Universal Robots PolyScope program: mt.urp

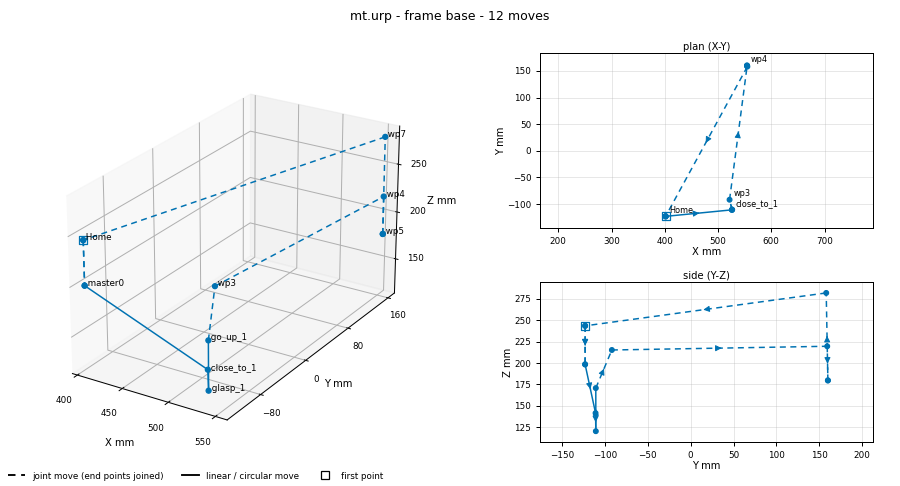
[picture p0: tool path of mt.urp in frame base, 12 of 12 moves have a stored position in this frame; points joined in program order, loops and branches not executed]
Program mt (installation=default directory=/programs/rovi createdIn=3.8.0.61336 lastSavedIn=3.8.0.61336 robotSerialNumber=2016352774)
Calibrated DH parameters: a=[0.000165, -0.326475, -0.363587, -0.000196, 0.000314, 0]; d=[0.089242, 611.192012, -553.715229, -57.366527, 0.094858, 0.082351]; alpha=[1.570545, 0.000446, 0.002569, 1.569839, -1.569769, 0]; deltaTheta=[-0.000028, 0.695517, -0.309849, -0.385645, -0.000052, -0.000026]
Robot Program (runOnlyOnce=false)
  MoveJ speed 60 deg/s, acceleration 80 deg/s^2 (useActiveTCP=false)
    Waypoint Home: TCP in base x=401.617 y=-123.055 z=243.432 mm, rx=-0.302 ry=3.1208 rz=0.0289 rad; joints [-1.945, -85.366, -123.205, -61.282, 91.24, -13.048] deg; flange x=401.666 y=-123.045 z=243.433 mm, rx=-2.4115 ry=1.9862 rz=0.0137 rad
  Loop Forever
    Script file /programs/X0.script
      | address="172.16.58.34"
      | port=3000
      | socket_open(address,port)
      | socket_send_line("X0()")
      | ret=socket_read_line(timeout=3)
      | socket_close()
    SuppressedNode
      MoveJ speed 60 deg/s, acceleration 80 deg/s^2 (useActiveTCP=false)
        Waypoint capture0: TCP in base x=291.074 y=-404.604 z=201.943 mm, rx=-1.3664 ry=-2.7229 rz=0.0094 rad; joints [-41.118, -99.563, -113.852, -61.83, 88.448, 12.2] deg
    MoveJ speed 60 deg/s, acceleration 80 deg/s^2 (useActiveTCP=false)
      Waypoint master0: TCP in base x=401.618 y=-123.109 z=198.453 mm, rx=-0.3017 ry=3.1209 rz=0.0292 rad; joints [-1.958, -89.361, -127.245, -53.252, 91.245, -13.033] deg; flange x=401.667 y=-123.1 z=198.454 mm, rx=-2.4113 ry=1.9864 rz=0.0139 rad
      Wait Sleep waitTime=0.5
    X_error := True
    Loop While (checkContinuously=false) expression=X_error
      Loop While (checkContinuously=false) expression=X_error
        Script file /programs/X1.script
          | address="172.16.58.34"
          | port=3000
          | X_error=False
          | socket_open(address,port)
          | p=get_actual_tcp_pose()
          | rpy=rotvec2rpy([p[3],p[4],p[5]])
          | socket_send_string("X1(")
          | socket_send_string(p[0])
          | socket_send_string(",")
          | socket_send_string(p[1])
          | socket_send_string(",")
          | socket_send_string(p[2])
          | socket_send_string(",")
          | socket_send_string(r2d(rpy[0]))
          | socket_send_string(",")
          | socket_send_string(r2d(rpy[1]))
          | socket_send_string(",")
          | socket_send_string(r2d(rpy[2]))
          | socket_send_line(")")
          | ret=socket_read_line(timeout=10)
          | if (ret!="OK"):
          |   X_error=True
          |   code=socket_read_string()
          |   popup(code,title="X1",blocking=True)
          | end
          | socket_close()
        Wait Sleep waitTime=0.5
      Script file /programs/rovi/X2.script
        | global X_var=Base
        | address="172.16.58.34"
        | port=3000
        | X_error=False
        | socket_open(address,port)
        | socket_send_line("X2()")
        | ret=socket_read_line(timeout=10)
        | if (ret != "OK"):
        |   X_error=True
        |   socket_close()
        | else:
        |   f=socket_read_ascii_float(6)
        |   while (f[0]!=6):
        |     sleep(0.3)
        |     f=socket_read_ascii_float(6)
        |   end
        |   socket_close()
        |   #popup(f,title="OK",blocking=True)
        |   rvec=rpy2rotvec([d2r(f[4]),d2r(f[5]),d2r(f[6])])
        |   counter=0
        |   while (counter<3):
        |     X_var[counter]=f[counter+1]
        |     counter=counter+1
        |   end
        |   counter=0
        |   while (counter<3):
        |     X_var[counter+3]=rvec[counter]
        |     counter=counter+1
        |   end
        | end
    Base := X_var
    MoveL speed 250 mm/s, acceleration 1200 mm/s^2 (useActiveTCP=false) feature(featureName=Joint_0_name)
      Waypoint close_to_1: TCP in base x=525.892 y=-110.922 z=141.644 mm, rx=-0.0249 ry=3.1389 rz=0.0305 rad; joints [-0.174, -109.589, -113.105, -47.241, 91.26, -1.103] deg; flange x=525.942 y=-110.921 z=141.644 mm, rx=-2.2278 ry=2.193 rz=0.0188 rad
      Waypoint glasp_1: TCP in base x=526.359 y=-110.603 z=120.526 mm, rx=-0.0225 ry=3.1387 rz=0.0305 rad; joints [-0.14, -111.796, -114.027, -44.096, 91.259, -0.976] deg
      Waypoint go_up_1: TCP in base x=526.461 y=-110.629 z=170.827 mm, rx=-0.0309 ry=3.1386 rz=0.0301 rad; joints [-0.138, -106.888, -111.412, -51.62, 91.249, -1.298] deg; flange x=526.511 y=-110.628 z=170.827 mm, rx=-2.232 ry=2.1887 rz=0.0182 rad
    MoveJ speed 60 deg/s, acceleration 80 deg/s^2 (useActiveTCP=false)
      Waypoint wp3: TCP in base x=521.639 y=-91.889 z=215.25 mm, rx=0.1315 ry=-3.1327 rz=-0.029 rad; joints [1.934, -102.24, -109.536, -58.64, 91.208, -2.926] deg; flange x=521.689 y=-91.885 z=215.25 mm, rx=-2.306 ry=2.1204 rz=0.0272 rad
      Waypoint wp4: TCP in base x=554.629 y=159.317 z=219.592 mm, rx=0.0228 ry=-3.1347 rz=-0.0286 rad; joints [26.953, -107.73, -101.658, -60.547, 91.26, 26.066] deg; flange x=554.679 y=159.318 z=219.591 mm, rx=-2.2315 ry=2.1995 rz=0.0276 rad
      Waypoint wp5: TCP in base x=554.357 y=160.095 z=179.72 mm, rx=0.0229 ry=-3.1347 rz=-0.0286 rad; joints [27.033, -110.662, -104.375, -54.897, 91.26, 26.156] deg; flange x=554.407 y=160.096 z=179.72 mm, rx=-2.2316 ry=2.1994 rz=0.0276 rad
      Waypoint wp6: TCP in base x=554.363 y=160.071 z=179.768 mm, rx=0.0228 ry=-3.1348 rz=-0.0288 rad; joints [27.031, -110.657, -104.374, -54.896, 91.262, 26.159] deg; flange x=554.413 y=160.072 z=179.767 mm, rx=-2.2314 ry=2.1994 rz=0.0276 rad
      Waypoint wp7: TCP in base x=555.075 y=158.144 z=281.8 mm, rx=0.0225 ry=-3.1348 rz=-0.0287 rad; joints [26.83, -104.167, -96.365, -69.405, 91.26, 25.931] deg; flange x=555.125 y=158.145 z=281.8 mm, rx=-2.2313 ry=2.1997 rz=0.0276 rad
    MoveJ speed 60 deg/s, acceleration 80 deg/s^2 (useActiveTCP=false)
      Waypoint Home: TCP in base x=401.617 y=-123.055 z=243.432 mm, rx=-0.302 ry=3.1208 rz=0.0289 rad; joints [-1.945, -85.366, -123.205, -61.282, 91.24, -13.048] deg; flange x=401.666 y=-123.045 z=243.433 mm, rx=-2.4115 ry=1.9862 rz=0.0137 rad
  Halt
  Folder Manual operation
    MoveJ speed 60 deg/s, acceleration 80 deg/s^2 (useActiveTCP=false)
      Waypoint master0: TCP in base x=401.618 y=-123.109 z=198.453 mm, rx=-0.3017 ry=3.1209 rz=0.0292 rad; joints [-1.958, -89.361, -127.245, -53.252, 91.245, -13.033] deg; flange x=401.667 y=-123.1 z=198.454 mm, rx=-2.4113 ry=1.9864 rz=0.0139 rad
    Base := Base
    Script file /programs/rovi/X0.script
      | address="172.16.58.34"
      | port=3000
      | socket_open(address,port)
      | socket_send_line("X0()")
      | ret=socket_read_line(timeout=3)
      | socket_close()
      | Base=p[0,0,0,0,0,0]
    Script file /programs/rovi/X1.script
      | address="172.16.58.34"
      | port=3000
      | timeout=10
      | socket_open(address,port)
      | p=get_actual_tcp_pose()
      | rpy=rotvec2rpy([p[3],p[4],p[5]])
      | socket_send_string("X1(")
      | socket_send_string(p[0])
      | socket_send_string(",")
      | socket_send_string(p[1])
      | socket_send_string(",")
      | socket_send_string(p[2])
      | socket_send_string(",")
      | socket_send_string(r2d(rpy[0]))
      | socket_send_string(",")
      | socket_send_string(r2d(rpy[1]))
      | socket_send_string(",")
      | socket_send_string(r2d(rpy[2]))
      | socket_send_line(")")
      | ret=socket_read_line(timeout=10)
      | if (ret!="OK"):
      |   code=socket_read_string()
      |   popup(code,title="X1",blocking=True)
      | end
      | socket_close()
